Staubli VAL3: start.pgx

public program start()
begin
  // Program Prog1 start
  // Program generated by RoboDK v3.8.4 for Staubli RX160 on 22/07/2019 15:36:39
  // Using nominal kinematics.
  nTraj=movej(jJoint[0],flange[0],mNomSpeed)
  nTraj=movej(jJoint[1],flange[0],mNomSpeed)
  nTraj=movel(pPoint[0],flange[0],mNomSpeed)
  nTraj=movec(pPoint[1],pPoint[2],flange[0],mNomSpeed)
  popUpMsg("Display message")
  delay(0.500)
  //call prog:Program1()
  do5=true
  WAIT FOR di5==true TIMEOUT=5000.0

  waitEndMove()
  // Program Prog1 end

end
